PROGRAM SFC
VAR
	Target: ARRAY [1..5] OF STRING := ['HOME','PosA','PosB','PosC','PosD'];
    TargIndex: INT:=0;
	qxGreenLamp :BOOL;
	qxRedLamp :BOOL;
	ElepseTime : TIME;
	TON_Blink1: TON;
	TON_Blink0: TON;
	Invisible: BOOL;
	MovingLamp: BOOL;
	ResetMemory : BOOl;
	TON_Moving: TON;
END_VAR

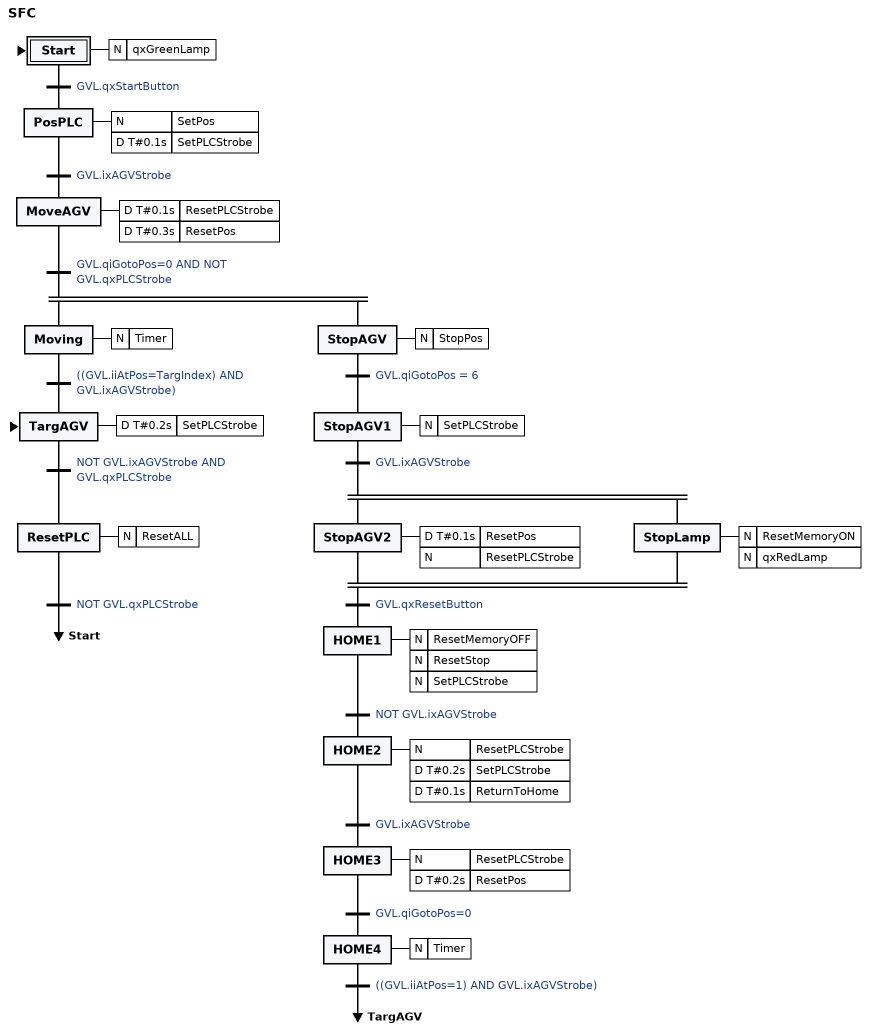
INITIAL_STEP Start:
    qxGreenLamp(N);
END_STEP
TRANSITION FROM Start TO PosPLC
    := GVL.qxStartButton;
END_TRANSITION
STEP PosPLC:
    SetPos(N);
    SetPLCStrobe(D, T#0.1s);
END_STEP
TRANSITION FROM PosPLC TO MoveAGV
    := GVL.ixAGVStrobe;
END_TRANSITION
STEP MoveAGV:
    ResetPLCStrobe(D, T#0.1s);
    ResetPos(D, T#0.3s);
END_STEP
TRANSITION FROM MoveAGV TO (Moving, StopAGV)
    := GVL.qiGotoPos=0 AND NOT GVL.qxPLCStrobe;
END_TRANSITION
STEP Moving:
    Timer(N);
END_STEP
STEP StopAGV:
    StopPos(N);
END_STEP
TRANSITION FROM StopAGV TO StopAGV1
    := GVL.qiGotoPos = 6;
END_TRANSITION
STEP StopAGV1:
    SetPLCStrobe(N);
END_STEP
TRANSITION FROM StopAGV1 TO (StopAGV2, StopLamp)
    := GVL.ixAGVStrobe;
END_TRANSITION
STEP StopAGV2:
    ResetPos(D, T#0.1s);
    ResetPLCStrobe(N);
END_STEP
STEP StopLamp:
    ResetMemoryON(N);
    qxRedLamp(N);
END_STEP
TRANSITION FROM (StopAGV2, StopLamp) TO HOME1
    := GVL.qxResetButton;
END_TRANSITION
STEP HOME1:
    ResetMemoryOFF(N);
    ResetStop(N);
    SetPLCStrobe(N);
END_STEP
TRANSITION FROM HOME1 TO HOME2
    := NOT GVL.ixAGVStrobe;
END_TRANSITION
STEP HOME2:
    ResetPLCStrobe(N);
    SetPLCStrobe(D, T#0.2s);
    ReturnToHome(D, T#0.1s);
END_STEP
TRANSITION FROM HOME2 TO HOME3
    := GVL.ixAGVStrobe;
END_TRANSITION
STEP HOME3:
    ResetPLCStrobe(N);
    ResetPos(D, T#0.2s);
END_STEP
TRANSITION FROM HOME3 TO HOME4
    := GVL.qiGotoPos=0;
END_TRANSITION
STEP HOME4:
    Timer(N);
END_STEP
TRANSITION FROM HOME4 TO TargAGV
    := ((GVL.iiAtPos=1) AND GVL.ixAGVStrobe);
END_TRANSITION
TRANSITION FROM Moving TO TargAGV
    := ((GVL.iiAtPos=TargIndex) AND GVL.ixAGVStrobe);
END_TRANSITION
STEP TargAGV:
    SetPLCStrobe(D, T#0.2s);
END_STEP
TRANSITION FROM TargAGV TO ResetPLC
    := NOT GVL.ixAGVStrobe AND GVL.qxPLCStrobe;
END_TRANSITION
STEP ResetPLC:
    ResetALL(N);
END_STEP
TRANSITION FROM ResetPLC TO Start
    := NOT GVL.qxPLCStrobe;
END_TRANSITION
// branch label Stop
// branch label MoveB

ACTION ResetALL:
GVL.qxPLCStrobe := FALSE;
GVL.qxStartButton := FALSE;
GVL.qxResetButton := FALSE;
GVL.qxStopButton := FALSE;
END_ACTION

ACTION ResetMemoryOFF:
ResetMemory := FALSE;
END_ACTION

ACTION ResetMemoryON:

ResetMemory := TRUE ;
END_ACTION

ACTION ResetPLCStrobe:
GVL.qxPLCStrobe := FALSE;
END_ACTION

ACTION ResetPos:
Gvl.qiGotoPos := 0;
END_ACTION

ACTION ResetStart:
GVL.qxStartButton :=FALSE;
END_ACTION

ACTION ResetStop:
GVL.qxStopButton := FALSE;
END_ACTION

ACTION ResetTarg:
TargIndex :=0;
END_ACTION

ACTION ReturnToHome:
GVL.qiGotoPos := 1;
GVL.qxResetButton := FALSE;
END_ACTION

ACTION SetPLCStrobe:
GVL.qxPLCStrobe := TRUE;
END_ACTION

ACTION SetPos:
GVL.qiGotoPos := TargIndex;
GVL.qxStartButton := FALSE;
END_ACTION

ACTION StopPos:
IF GVL.qxStopButton THEN
	GVL.qiGotoPos := 6;
END_IF
END_ACTION

ACTION Timer:
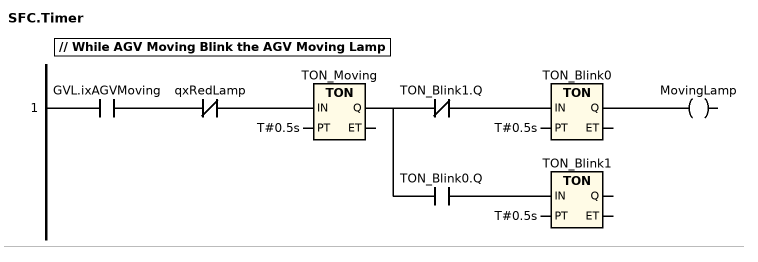
// NETWORK 1
// label: // While AGV Moving Blink the AGV Moving Lamp
TON_Moving(IN := GVL.ixAGVMoving AND NOT qxRedLamp, PT := T#0.5s); // TON
TON_Blink0(IN := TON_Moving.Q AND NOT TON_Blink1.Q, PT := T#0.5s); // TON
MovingLamp := TON_Blink0.Q;
TON_Blink1(IN := TON_Moving.Q AND TON_Blink0.Q, PT := T#0.5s); // TON
END_ACTION

END_PROGRAM

(* stored: Version 1.1.0.1, ProductVersion 3.1.4024.12
   POU SFC: Id {cb8d6808-a441-40b3-8b65-f09fd5dd5a2a}, SpecialFunc None
   Action ResetALL: Id {ecad7b1c-2b17-4714-ac18-04dab0034184}
   Action ResetMemoryOFF: Id {9bc50f40-a656-49ce-a16c-4a49181017fc}
   Action ResetMemoryON: Id {aa823f5f-5ff2-4d30-a56c-12d7863b6f50}
   Action ResetPLCStrobe: Id {33f727d1-1014-42d8-8b65-899e4d78ced6}
   Action ResetPos: Id {7bdd900d-1a24-45d5-8f97-dac9e89031a8}
   Action ResetStart: Id {e3b30ba5-97a6-41b2-add1-72103aca92e8}
   Action ResetStop: Id {122a0584-6b15-4f4d-b96a-b942b3c7e242}
   Action ResetTarg: Id {7359be6d-4eae-45ea-803e-216e260620f7}
   Action ReturnToHome: Id {4cf96541-038b-4b0f-a38f-6a7eccafac94}
   Action SetPLCStrobe: Id {48c40871-58e2-47c8-a541-33b31745a6c1}
   Action SetPos: Id {5e206b8f-6b07-47e6-bd41-ec0a628f022d}
   Action StopPos: Id {9626d84e-652c-43e2-ae72-839241b56827}
   Action Timer: Id {80282cf6-a21f-49db-a647-bd8eeabdc4ea} *)
